// TIA Portal V17 export
// export: Created 2023-06-23T18:33:38.8781423Z, ExportSetting WithDefaults, DisplayName Totally Integrated Automation Portal, DisplayVersion V17, DisplayName TIA Portal Openness, DisplayVersion V17, DisplayName TIA Portal Version Control Interface, DisplayVersion V17, DisplayName STEP 7 Professional, DisplayVersion V17, DisplayName STEP 7 Safety, DisplayVersion V17, DisplayName WinCC Advanced / Unified PC, DisplayVersion V17
VAR_GLOBAL   // PLC tag table "12_PL-1"
   "iPL-1" AT %I8.4 : Bool;
   "oPL-1" AT %Q1.1 : Bool;
END_VAR
